FUNCTION read_2bytes : INT
VAR_INPUT
	gvl_highbyte : BYTE;
	gvl_lowbyte : BYTE;
	
END_VAR
VAR
	//value : INT; 
	p_value : HighLow_pointers; 
END_VAR

p_value.pLow_byte := ADR(read_2bytes);
p_value.pHigh_byte := p_value.pLow_byte +1;
p_value.pLow_byte^ := gvl_lowbyte;
p_value.pHigh_byte^ := gvl_highbyte;

END_FUNCTION

(* stored: Version 1.1.0.1, ProductVersion 3.1.4024.9
   POU read_2bytes: Id {881ad0ad-5a88-4ee2-9f76-6e46b6b8049a}, SpecialFunc None *)
